Yaskawa INFORM job: u_incl_braA1.JBI

/JOB
//NAME u_incl_braA1
///FOLDERNAME DEMO
//POS
///NPOS 0,0,0,0,0,0
///TOOL 7
///POSTYPE ROBOT
///RECTAN
///RCONF 1,0,0,0,0,0,0,0,0,0,0,0,0,0,0,0,0,0,0,0,0,0,0,0
//INST
///DATE 2021/02/10 13:51
///COMM
///ATTR SC,RW,RJ
////FRAME USER 2
///GROUP1 RB1
///GROUP2 ST1
NOP
CALL JOB:DEBUT
'Part trajectory number: 0
CALL JOB:u_incl_braA1TRJ0
CALL JOB:FIN
END
